// TIA Portal V17 export
// export: Created 2023-12-22T15:03:18.8862502Z, ExportSetting WithDefaults, DisplayName Totally Integrated Automation Portal, DisplayVersion V17, DisplayName TIA Portal Openness, DisplayVersion V17, DisplayName TIA Portal Version Control Interface, DisplayVersion V17, DisplayName STEP 7 Professional, DisplayVersion V17, DisplayName STEP 7 Safety, DisplayVersion V17, DisplayName WinCC Advanced, DisplayVersion V17
DATA_BLOCK "Comm_Scada"   // DB9
{ S7_Optimized_Access := 'FALSE' }
VERSION : 0.1
// stored: AutoNumber false, DBAccessibleFromOPCUA true, DBAccessibleFromWebserver true, IsOnlyStoredInLoadMemory false, IsWriteProtectedInAS false
   VAR
      Input : Struct
         LE_105_Result : Real;
         LE_106_Result : Real;
         LE_107_Result : Real;
         LE_108_Result : Real;
         TE_101_Result : Real;
         TE_102_Result : Real;
         TE_103_Result : Real;
         TE_104_Result : Real;
         LE_105_Alarm : Word;
         LE_106_Alarm : Word;
         LE_107_Alarm : Word;
         LE_108_Alarm : Word;
         TE_101_Alarm : Word;
         TE_102_Alarm : Word;
         TE_103_Alarm : Word;
         TE_104_Alarm : Word;
         rez_1 : Word;
         rez_2 : Word;
         rez_3 : Word;
         rez_4 : Word;
         rez_5 : Word;
      END_STRUCT;
      Output : Struct
         rez_1 : Word;
         rez_2 : Word;
         rez_3 : Word;
         rez_4 : Word;
         rez_5 : Word;
      END_STRUCT;
   END_VAR
BEGIN
END_DATA_BLOCK
